FUNCTION TryConvert_BYTE_TO_BYTE : BOOL
VAR_INPUT
	in : BYTE;
	out : REFERENCE TO BYTE;
END_VAR

out := in;
TryConvert_BYTE_TO_BYTE := TRUE;

END_FUNCTION

(* stored: Version 1.1.0.1, ProductVersion 3.1.4024.12
   POU TryConvert_BYTE_TO_BYTE: Id {3276fd64-33c4-4c68-afeb-b59294632005}, SpecialFunc None *)
